KUKA KRL data list: separa.dat

&ACCESS RV
DEFDAT separa PUBLIC

ENDDAT
